{attribute 'GeneratedUsingTerminal: EK1100-0000-0018'}
{attribute addProperty BoxType "EK1100-0000-0018"}
{attribute addProperty Id "RC30_B1_EL7041_1000EL7041_86DE63E743RC30_B2_EL7041_1000EL7041_86DE63E743RC30_C11_EL7041_1000EL7041_86DE63E743RC30_C12_EL7041_1000EL7041_86DE63E743RC30_C21_EL7041_1000EL7041_86DE63E743RC30_C22_EL7041_1000EL7041_86DE63E743RC30_2_EndTerminal_EL9010EL9010_D29C20850"}
{attribute addProperty CRC "2316296572"}
{attribute addProperty Size "258"}
{attribute addProperty Name "RC30_2 (EK1100)"}
TYPE RC30_2_EK1100_8A0FE17C EXTENDS EK1100_1FC0878B :
STRUCT
	{attribute addProperty Name "RC30_B1 (EL7041-1000)"}
	{attribute addProperty PreviousPort "RC30_2 (EK1100) : B"}
	{attribute addProperty SyncUnit "C30"}
	RC30_B1_EL7041_1000 : EL7041_86DE63E7;
	{attribute addProperty Name "RC30_B2 (EL7041-1000)"}
	{attribute addProperty PreviousPort "RC30_B1 (EL7041-1000) : B"}
	{attribute addProperty SyncUnit "C30"}
	RC30_B2_EL7041_1000 : EL7041_86DE63E7;
	{attribute addProperty Name "RC30_C11 (EL7041-1000)"}
	{attribute addProperty PreviousPort "RC30_B2 (EL7041-1000) : B"}
	{attribute addProperty SyncUnit "C30"}
	RC30_C11_EL7041_1000 : EL7041_86DE63E7;
	{attribute addProperty Name "RC30_C12 (EL7041-1000)"}
	{attribute addProperty PreviousPort "RC30_C11 (EL7041-1000) : B"}
	{attribute addProperty SyncUnit "C30"}
	RC30_C12_EL7041_1000 : EL7041_86DE63E7;
	{attribute addProperty Name "RC30_C21 (EL7041-1000)"}
	{attribute addProperty PreviousPort "RC30_C12 (EL7041-1000) : B"}
	{attribute addProperty SyncUnit "C30"}
	RC30_C21_EL7041_1000 : EL7041_86DE63E7;
	{attribute addProperty Name "RC30_C22 (EL7041-1000)"}
	{attribute addProperty PreviousPort "RC30_C21 (EL7041-1000) : B"}
	{attribute addProperty SyncUnit "C30"}
	RC30_C22_EL7041_1000 : EL7041_86DE63E7;
	{attribute addProperty Name "RC30_2_EndTerminal (EL9010)"}
	{attribute addProperty PreviousPort "RC30_C22 (EL7041-1000) : B"}
	{attribute addProperty SyncUnit "default"}
	RC30_2_EndTerminal_EL9010 : EL9010_D29C2085;
END_STRUCT
END_TYPE

(* stored: Version 1.2.0.0, ProductVersion 3.1.4024.11
   DUT RC30_2_EK1100_8A0FE17C: Id {8879c74c-785b-00b9-3fa3-8b1b5a6ac1a2} *)
